% RSLogix 500 project ML1100S9.RSS, saved by version 8.10.00.18 %
PROJECT "UNTITLED"    % processor: Bul.1763 MicroLogix 1100 Series A %

PROGRAM FILES
  LAD 2   9 rungs

DATA FILES
  O0 OUTPUT  6 elements
  I1 INPUT  12 elements
  S2 STATUS  66 elements
  B3 BINARY  1 elements
  T4 TIMER  1 elements
  C5 COUNTER  1 elements
  R6 CONTROL  1 elements
  N7 INTEGER  10 elements
  F8 FLOAT  1 elements

LADDER 2
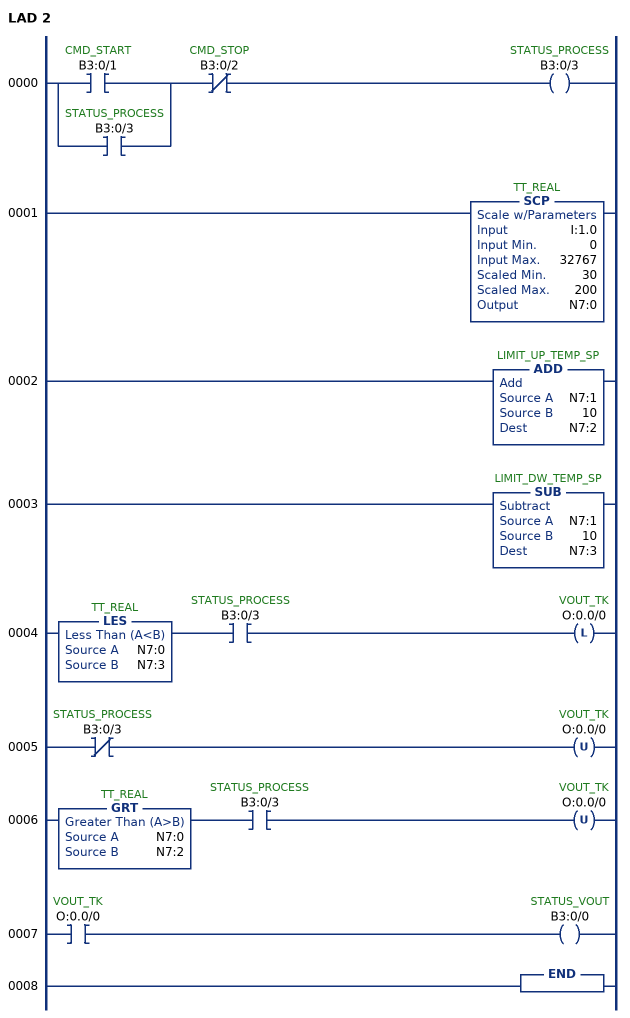
% Rung: 0 %
SOR BST XIC B3:0/1 NXB XIC B3:0/3 BND XIO B3:0/2 OTE B3:0/3 EOR
%   B3:0/1  CMD_START %
%   B3:0/3  STATUS_PROCESS %
%   B3:0/2  CMD_STOP %
% Rung: 1 %  % edit flag set %
SOR SCP I:1.0 0 32767 30 200 N7:0 EOR
%   I:1.0  TT_INT %
%   N7:0  TT_REAL %
% Rung: 2 %
SOR ADD N7:1 10 N7:2 EOR
%   N7:1  CMD_TEMP_SP %
%   N7:2  LIMIT_UP_TEMP_SP %
% Rung: 3 %
SOR SUB N7:1 10 N7:3 EOR
%   N7:1  CMD_TEMP_SP %
%   N7:3  LIMIT_DW_TEMP_SP %
% Rung: 4 %
SOR LES N7:0 N7:3 XIC B3:0/3 OTL O:0.0/0 EOR
%   N7:0  TT_REAL %
%   N7:3  LIMIT_DW_TEMP_SP %
%   B3:0/3  STATUS_PROCESS %
%   O:0.0/0  VOUT_TK %
% Rung: 5 %
SOR XIO B3:0/3 OTU O:0.0/0 EOR
%   B3:0/3  STATUS_PROCESS %
%   O:0.0/0  VOUT_TK %
% Rung: 6 %
SOR GRT N7:0 N7:2 XIC B3:0/3 OTU O:0.0/0 EOR
%   N7:0  TT_REAL %
%   N7:2  LIMIT_UP_TEMP_SP %
%   B3:0/3  STATUS_PROCESS %
%   O:0.0/0  VOUT_TK %
% Rung: 7 %
SOR XIC O:0.0/0 OTE B3:0/0 EOR
%   O:0.0/0  VOUT_TK %
%   B3:0/0  STATUS_VOUT %
% Rung: 8 %
SOR END EOR

OTHER DOCUMENTED ADDRESSES
  I:0.0/0  IN_START
  I:0.0/1  IN_STOP
